FUNCTION_BLOCK FB_ModuleBase EXTENDS FB_PackMLModeSet
VAR_INPUT
	ModuleCtrl : REFERENCE TO ST_ModuleCtrl;
	SystemContext : REFERENCE TO ST_SystemContext;
	HeartbeatIndex : UDINT;
	RuntimeConfig : REFERENCE TO ST_ModuleRuntimeConfig;
	VariableNodeReader : I_VariableNodeReader;
END_VAR

VAR_OUTPUT
	ModuleStatus : ST_ModuleStatus;
	ModuleVariableList : ARRAY[1..Param_Config.MaxModuleVariable] OF ST_ExtDescriptor;
	ModuleAlarmList : ARRAY[1..Param_Config.MaxPublishedModuleAlarms] OF ST_ExtAlarm;
	ModuleDataList : ARRAY[1..Param_Config.MaxModuleData] OF ST_ExtDescriptor;
END_VAR

VAR
	_CmdRequestOneShot : R_TRIG;
	_ModeRequestOneShot : R_TRIG;
	
	_ModuleId : UDINT;
	_ServiceContext : ST_ServiceContext;
	
	_HeartbeatTimer : TON;
	_LastHeartbeatIndex : UDINT;
	_IsControlSourceAlive : BOOL;
	_ConfiguredSnapshot : FB_ConfigValueSnapshotReader;
	_AlarmManager : FB_ModuleAlarmManager;
	_InAlarmHook : BOOL;
	_InVariableHook : BOOL;
	_ConfiguredVariableCount : UINT;
	_ServiceCoordinator : FB_ServiceCoordinator;
	_ServiceRegistrationAttempted : BOOL;
END_VAR

METHOD PROTECTED FINAL H_OnAborting : E_PackMLHookResult
VAR_INPUT
	bFirstScan : BOOL;
END_VAR
H_OnAborting := E_PackMLHookResult.Busy;
IF _ServiceCoordinator.AllAborted THEN
	H_OnAborting := E_PackMLHookResult.Done;
END_IF
END_METHOD

METHOD PROTECTED FINAL H_OnClearing : E_PackMLHookResult
VAR_INPUT
	bFirstScan : BOOL;
END_VAR
H_OnClearing := E_PackMLHookResult.Busy;
IF _ServiceCoordinator.AllStopped THEN
	H_OnClearing := E_PackMLHookResult.Done;
END_IF
END_METHOD

METHOD PROTECTED FINAL H_OnIdle
VAR_INPUT
	bFirstScan	: BOOL;
END_VAR
// Transfer to execute automatically
RequestCommand(E_PackMLCommand.Start);
END_METHOD

METHOD PROTECTED FINAL H_OnResetting : E_PackMLHookResult
VAR_INPUT
	bFirstScan : BOOL;
END_VAR
H_OnResetting := E_PackMLHookResult.Busy;
IF _ServiceCoordinator.AllIdle THEN
	H_OnResetting := E_PackMLHookResult.Done;
END_IF
END_METHOD

METHOD PROTECTED FINAL H_OnStopping : E_PackMLHookResult
VAR_INPUT
	bFirstScan : BOOL;
END_VAR
H_OnStopping := E_PackMLHookResult.Busy;
IF _ServiceCoordinator.AllStopped THEN
	H_OnStopping := E_PackMLHookResult.Done;
END_IF
END_METHOD

METHOD PROTECTED H_RegisterServices
// Derived Modules register persistent Service storage once.
END_METHOD

METHOD PROTECTED H_UpdateAlarm
// Optional Module extension; submitted values belong to this scan.
END_METHOD

METHOD PROTECTED H_UpdateBaseUnit
VAR_INPUT
END_VAR
END_METHOD

METHOD PROTECTED H_UpdateService
VAR_INPUT
END_VAR
END_METHOD

METHOD PROTECTED H_UpdateVariable
// Optional Module extension; submitted values belong to this scan.
END_METHOD

METHOD PROTECTED FINAL M_AddAlarm : BOOL
VAR_INPUT
	MainErrorId : UDINT;
	SourceErrorId : UDINT;
	Message : STRING;
	Path : STRING(255);
	Severity : E_Severity;
END_VAR
VAR
	nIndex : UINT;
	Alarm : ST_ExtAlarm;
END_VAR
M_AddAlarm := FALSE;
IF NOT _InAlarmHook OR (MainErrorId = 0) THEN
	RETURN;
END_IF
IF __ISVALIDREF(RuntimeConfig) THEN
	IF RuntimeConfig.Valid THEN
		FOR nIndex := 1 TO RuntimeConfig.AlarmCount DO
			IF RuntimeConfig.AlarmBindings[nIndex].Definition.MainErrorId = MainErrorId THEN
				M_AddAlarm := TRUE; // JSON owns the complete definition, even without a valid sample.
				RETURN;
			END_IF
		END_FOR
	END_IF
END_IF
MEMSET(ADR(Alarm), 0, SIZEOF(Alarm));
Alarm.MainErrorId := MainErrorId;
Alarm.SourceErrorId := SourceErrorId;
Alarm.Message := Message;
Alarm.Path := Path;
Alarm.Severity := Severity;
Alarm.DateTime := _ServiceContext.UtcDateTime;
M_AddAlarm := _AlarmManager.M_ObserveHookAlarm(Alarm := Alarm);
END_METHOD

METHOD PROTECTED FINAL M_AddVariable : BOOL
VAR_INPUT
	Id : UDINT;
	Name : STRING(30);
	DataType : E_DescriptorType;
	Unit : STRING(10);
	Value : STRING(80);
END_VAR
VAR
	nIndex : UINT;
END_VAR
M_AddVariable := FALSE;
IF NOT _InVariableHook OR (Id = 0) THEN
	RETURN;
END_IF
FOR nIndex := 1 TO ModuleStatus.Variable.PublishedCount DO
	IF ModuleVariableList[nIndex].Id = Id THEN
		IF nIndex <= _ConfiguredVariableCount THEN
			M_AddVariable := TRUE; // JSON ownership is not a duplicate submission.
		ELSIF ModuleStatus.Variable.DuplicateId = 0 THEN
			ModuleStatus.Variable.DuplicateId := Id;
		END_IF
		RETURN;
	END_IF
END_FOR
IF ModuleStatus.Variable.PublishedCount >= Param_Config.MaxModuleVariable THEN
	ModuleStatus.Variable.Overflow := TRUE;
	RETURN;
END_IF
ModuleStatus.Variable.PublishedCount := ModuleStatus.Variable.PublishedCount + 1;
nIndex := ModuleStatus.Variable.PublishedCount;
ModuleVariableList[nIndex].Id := Id;
ModuleVariableList[nIndex].Name := Name;
ModuleVariableList[nIndex].DataType := DataType;
ModuleVariableList[nIndex].Unit := Unit;
ModuleVariableList[nIndex].Value := Value;
M_AddVariable := TRUE;
END_METHOD

METHOD PRIVATE M_CheckHeartbeat
VAR_INPUT
END_VAR

VAR
	bLooseHeartbeat : BOOL;
	HeartbeatTimeout : TIME;
END_VAR
HeartbeatTimeout := SystemContext.ModuleHeartbeatTimeout;
IF HeartbeatTimeout <= T#0S THEN
	HeartbeatTimeout := Param_Config.ModuleHeartbeat_Timeout;
END_IF

// Heartbeats check
bLooseHeartbeat := _LastHeartbeatIndex = HeartbeatIndex;
IF bLooseHeartbeat THEN
	_HeartbeatTimer(IN := TRUE, PT := HeartbeatTimeout);
ELSE
	_HeartbeatTimer(IN := FALSE, PT := HeartbeatTimeout);
END_IF

// Update Last Heartbeat Index
_LastHeartbeatIndex := HeartbeatIndex;

// Update Is ControlSource Alive status
_IsControlSourceAlive := NOT _HeartbeatTimer.Q;
END_METHOD

METHOD PRIVATE M_PublishAlarmState
_AlarmManager.M_Publish(AlarmList := ModuleAlarmList);
ModuleStatus.Alarm.AckResponseId := _AlarmManager.AckResponseId;
ModuleStatus.Alarm.AckAccepted := _AlarmManager.AckAccepted;
ModuleStatus.Alarm.AckError := _AlarmManager.AckError;
ModuleStatus.Alarm.ConfiguredLatchedCount := _AlarmManager.ConfiguredLatchedCount;
ModuleStatus.Alarm.Overflow := _AlarmManager.Overflow;
ModuleStatus.Alarm.ServiceLatchedCount := _AlarmManager.ServiceLatchedCount;
ModuleStatus.Alarm.HookLatchedCount := _AlarmManager.HookLatchedCount;
ModuleStatus.Alarm.DuplicateId := _AlarmManager.DuplicateId;
END_METHOD

METHOD PROTECTED FINAL M_RegisterService : BOOL
VAR_INPUT
	ServiceId : UDINT;
	AllowCompositeCall : BOOL;
	UpperParam : ANY;
	EffectiveParam : ANY;
END_VAR
VAR_IN_OUT
	UpperCtrl : ST_ServiceCtrl;
	EffectiveCtrl : ST_ServiceCtrl;
	Status : ST_ServiceStatus;
END_VAR
M_RegisterService := _ServiceCoordinator.M_Register(
	ServiceId := ServiceId,
	AllowCompositeCall := AllowCompositeCall,
	UpperCtrl := UpperCtrl,
	EffectiveCtrl := EffectiveCtrl,
	UpperParam := UpperParam,
	EffectiveParam := EffectiveParam,
	Status := Status);
END_METHOD

METHOD PRIVATE M_UpdateAlarmState
VAR
	nAlarm : UINT;
	nSource : UINT;
	nRevision : UDINT;
	fValue : LREAL;
	bValid : BOOL;
	bConditionMet : BOOL;
	Alarm : ST_ExtAlarm;
END_VAR
nRevision := 0;
IF __ISVALIDREF(RuntimeConfig) THEN
	IF RuntimeConfig.Valid THEN
		nRevision := RuntimeConfig.Revision;
	END_IF
END_IF
_AlarmManager.M_BeginCycle(
	ModuleId := _ModuleId,
	ConfigurationRevision := nRevision);

// Remove identities now owned by JSON before an acknowledgement can find a stale Hook event.
IF __ISVALIDREF(RuntimeConfig) THEN
	IF RuntimeConfig.Valid THEN
		FOR nAlarm := 1 TO RuntimeConfig.AlarmCount DO
			_AlarmManager.M_SuppressHookAlarm(
				MainErrorId := RuntimeConfig.AlarmBindings[nAlarm].Definition.MainErrorId);
		END_FOR
	END_IF
END_IF

// Process acknowledgements before evaluating this cycle so AckAll cannot consume
// a new event that the upper controller has not observed yet.
_AlarmManager.M_ProcessAcknowledgement(Request := ModuleCtrl.AlarmAckRequest);

IF __ISVALIDREF(RuntimeConfig) THEN
	IF RuntimeConfig.Valid AND _ConfiguredSnapshot.Ready THEN
		FOR nAlarm := 1 TO RuntimeConfig.AlarmCount DO
			nSource := RuntimeConfig.VariableCount + nAlarm;
			fValue := _ConfiguredSnapshot.M_GetLReal(SourceIndex := nSource, Valid => bValid);
			bConditionMet := FALSE;
			IF bValid THEN
				bConditionMet := F_AlarmConditionMet(
					Value := fValue,
					Operator := RuntimeConfig.AlarmBindings[nAlarm].Definition.Operator,
					Threshold := RuntimeConfig.AlarmBindings[nAlarm].Definition.Threshold,
					Tolerance := RuntimeConfig.AlarmBindings[nAlarm].Definition.Tolerance);
			END_IF

			MEMSET(ADR(Alarm), 0, SIZEOF(Alarm));
			Alarm.ModuleId := _ModuleId;
			Alarm.ServiceId := 0;
			Alarm.MainErrorId := RuntimeConfig.AlarmBindings[nAlarm].Definition.MainErrorId;
			Alarm.SourceErrorId := RuntimeConfig.AlarmBindings[nAlarm].Definition.SourceErrorId;
			Alarm.Message := RuntimeConfig.AlarmBindings[nAlarm].Definition.Message;
			Alarm.Path := RuntimeConfig.AlarmBindings[nAlarm].Definition.Source;
			Alarm.Severity := RuntimeConfig.AlarmBindings[nAlarm].Definition.Severity;
			_AlarmManager.M_UpdateConfiguredAlarm(
				AlarmIndex := nAlarm,
				SampleValid := bValid,
				ConditionMet := bConditionMet,
				Alarm := Alarm,
				UtcDateTime := _ServiceContext.UtcDateTime);
		END_FOR
	END_IF
END_IF

_InAlarmHook := TRUE;
H_UpdateAlarm();
_InAlarmHook := FALSE;

M_UpdateServiceAlarms();
_AlarmManager.M_EndCycle();
END_METHOD

METHOD PRIVATE M_UpdateConfiguredVariableList
VAR
	nVariable : UINT;
	bValid : BOOL;
END_VAR
IF NOT __ISVALIDREF(RuntimeConfig) THEN
	RETURN;
END_IF
IF NOT RuntimeConfig.Valid THEN
	RETURN;
END_IF

FOR nVariable := 1 TO RuntimeConfig.VariableCount DO
	ModuleVariableList[nVariable].Id := RuntimeConfig.VariableBindings[nVariable].Definition.Id;
	ModuleVariableList[nVariable].Name := RuntimeConfig.VariableBindings[nVariable].Definition.Name;
	ModuleVariableList[nVariable].DataType := F_ConfigDataTypeToDescriptor(
		DataType := RuntimeConfig.VariableBindings[nVariable].Definition.DataType);
	ModuleVariableList[nVariable].Unit := RuntimeConfig.VariableBindings[nVariable].Definition.Unit;
	ModuleVariableList[nVariable].Value := _ConfiguredSnapshot.M_GetValueString(
		SourceIndex := nVariable,
		Valid => bValid);
END_FOR
_ConfiguredVariableCount := RuntimeConfig.VariableCount;
ModuleStatus.Variable.PublishedCount := _ConfiguredVariableCount;
END_METHOD

METHOD PROTECTED FINAL M_UpdateModule
IF NOT _ServiceRegistrationAttempted THEN
	_ServiceRegistrationAttempted := TRUE;
	_ServiceCoordinator.M_BeginRegistration();
	H_RegisterServices();
	_ServiceCoordinator.M_Seal();
END_IF

M_CheckHeartbeat();
ModuleStatus.IsControlSourceAlive := _IsControlSourceAlive;

// Update module state machine
PackMLIn := ModuleCtrl.PackMLIn;
SUPER^();

IF __ISVALIDREF(RuntimeConfig) THEN
	_ModuleId := RuntimeConfig.ModuleId;
	_ConfiguredSnapshot(
		RuntimeConfig := RuntimeConfig,
		VariableNodeReader := VariableNodeReader);
	ModuleStatus.ModuleId := _ModuleId;
	ModuleStatus.Enabled := RuntimeConfig.Enabled;
	ModuleStatus.ModuleType := RuntimeConfig.ModuleType;
END_IF

_ServiceContext.ModuleId := _ModuleId;
_ServiceContext.UtcDateTime := SystemContext.UtcDateTime;

// Update service state machine
_ServiceCoordinator.M_PrepareCycle(
	ModuleInExecute := PackMLOut.eStateCurrent = E_PackMLState.Execute,
	ModuleCtrl := ModuleCtrl);
H_UpdateService();

// Update base unit state machine
H_UpdateBaseUnit();

// Capture the status set produced by this scan for framework aggregation and
// for the Module PackML transition checks in the next scan.
_ServiceCoordinator.M_ObserveCycle();

_CmdRequestOneShot(CLK:= PackMLIn.bCommandChangeRequest, Q=> );
_ModeRequestOneShot(CLK:= PackMLIn.bModeChangeRequest, Q=> );

// Updata status
IF _CmdRequestOneShot.Q OR _ModeRequestOneShot.Q THEN
	ModuleStatus.ResponseId := ModuleCtrl.RequestId;
END_IF
ModuleStatus.PackMLOut := PackMLOut;

M_UpdateAlarmState();
M_PublishAlarmState();
M_UpdateServiceDataList();
M_UpdateVariableList();
END_METHOD

METHOD PRIVATE M_UpdateServiceAlarms
VAR
	nServiceIndex : UINT;
	nErrorIndex : UINT;
	ServiceStatus : ST_ServiceStatus;
END_VAR
// Submit currently observable Service errors. The manager owns lifecycle state
// and marks identities not observed in this scan inactive during M_EndCycle.
FOR nServiceIndex := 1 TO _ServiceCoordinator.RegisteredCount DO
	IF NOT _ServiceCoordinator.M_GetServiceStatusByIndex(
		Index := nServiceIndex,
		Status => ServiceStatus) THEN
		CONTINUE;
	END_IF
	FOR nErrorIndex := 1 TO Param_Config.MaxServiceError DO
		IF ServiceStatus.ErrorList[nErrorIndex].MainErrorId <> 0 THEN
			_AlarmManager.M_ObserveServiceAlarm(
				Alarm := ServiceStatus.ErrorList[nErrorIndex]);
		END_IF
	END_FOR
END_FOR
END_METHOD

METHOD PRIVATE M_UpdateServiceDataList
VAR
	nServiceIndex : UINT;
	nDataIndex : UINT;
	nPublishedIndex : UINT;
	bDuplicate : BOOL;
	DataId : UDINT;
	ServiceStatus : ST_ServiceStatus;
END_VAR
MEMSET(ADR(ModuleDataList), 0, SIZEOF(ModuleDataList));
MEMSET(ADR(ModuleStatus.Data), 0, SIZEOF(ModuleStatus.Data));

FOR nServiceIndex := 1 TO _ServiceCoordinator.RegisteredCount DO
	IF NOT _ServiceCoordinator.M_GetServiceStatusByIndex(
		Index := nServiceIndex,
		Status => ServiceStatus) THEN
		CONTINUE;
	END_IF
	IF ServiceStatus.Data.Overflow THEN
		ModuleStatus.Data.Overflow := TRUE;
	END_IF

	FOR nDataIndex := 1 TO Param_Config.MaxServiceData DO
		DataId := ServiceStatus.Data.DataList[nDataIndex].Id;
		IF DataId = 0 THEN
			CONTINUE;
		END_IF

		bDuplicate := FALSE;
		FOR nPublishedIndex := 1 TO ModuleStatus.Data.PublishedCount DO
			IF ModuleDataList[nPublishedIndex].Id = DataId THEN
				bDuplicate := TRUE;
				EXIT;
			END_IF
		END_FOR

		IF bDuplicate THEN
			IF ModuleStatus.Data.DuplicateId = 0 THEN
				ModuleStatus.Data.DuplicateId := DataId;
			END_IF
			CONTINUE;
		END_IF

		IF ModuleStatus.Data.PublishedCount >= Param_Config.MaxModuleData THEN
			ModuleStatus.Data.Overflow := TRUE;
			CONTINUE;
		END_IF

		ModuleStatus.Data.PublishedCount := ModuleStatus.Data.PublishedCount + 1;
		ModuleDataList[ModuleStatus.Data.PublishedCount] :=
			ServiceStatus.Data.DataList[nDataIndex];
	END_FOR
END_FOR
END_METHOD

METHOD PRIVATE M_UpdateVariableList
MEMSET(ADR(ModuleVariableList), 0, SIZEOF(ModuleVariableList));
MEMSET(ADR(ModuleStatus.Variable), 0, SIZEOF(ModuleStatus.Variable));
_ConfiguredVariableCount := 0;
M_UpdateConfiguredVariableList();
_InVariableHook := TRUE;
H_UpdateVariable();
_InVariableHook := FALSE;
END_METHOD

END_FUNCTION_BLOCK

(* stored: Version 1.1.0.1, ProductVersion 3.1.4026.18
   POU FB_ModuleBase: Id {6193009a-0dba-45cf-9862-8c04373cb73b}, SpecialFunc None
   Folder HookMethod: Id {0b542957-3892-4df2-b0e7-9c93700d86b5}
   Folder Private: Id {9fe464c1-8082-49c4-bb39-67807fabb98d}
   Folder StateAction: Id {11d8fc2a-f5c5-4f28-ab4c-743399b9bdc9}
   Method H_OnAborting: Id {8915d7ec-4b86-49c6-9413-c27372315251}
   Method H_OnClearing: Id {f0397c47-1f8c-451b-93d5-b31f3f0b03fb}
   Method H_OnIdle: Id {1f951a38-751e-4488-9f76-b0388bffa732}
   Method H_OnResetting: Id {9a955b11-d840-4734-887a-1f112a090756}
   Method H_OnStopping: Id {59c31d14-1773-47ac-a868-c25bd37caf0c}
   Method H_RegisterServices: Id {cfb22052-7349-4b72-a01d-2a1212d3d28d}
   Method H_UpdateAlarm: Id {cb61c708-0f3f-469b-a964-b4b351dc9538}
   Method H_UpdateBaseUnit: Id {cce9c8f5-b668-43c6-ab47-4d2999638c8f}
   Method H_UpdateService: Id {d906a778-6b57-49b8-9e25-ec7461c4759a}
   Method H_UpdateVariable: Id {9d15debf-7709-4c12-8971-2dc378590faa}
   Method M_AddAlarm: Id {7c4e4f34-fc5f-482d-9a72-920e07d0a35d}
   Method M_AddVariable: Id {669b3f9b-b87a-4c72-b049-e0b92818a4d4}
   Method M_CheckHeartbeat: Id {95356be4-c779-4a0a-84d9-ca5fd7d93bc1}
   Method M_PublishAlarmState: Id {055c5419-f6a5-46d2-bb31-19f68a24d121}
   Method M_RegisterService: Id {f7cafede-9912-44aa-8775-3dd24b828568}
   Method M_UpdateAlarmState: Id {6b9b6538-c160-4a7b-93a1-a430b340815a}
   Method M_UpdateConfiguredVariableList: Id {6e5b225f-a33a-409e-827d-1330e9e22088}
   Method M_UpdateModule: Id {a3ee927e-c27b-49bf-8f5e-1ddb1a222fc5}
   Method M_UpdateServiceAlarms: Id {aac9cb3d-dfbb-4fd3-8423-c48f0de4cb6b}
   Method M_UpdateServiceDataList: Id {09acfa8b-205a-4e4b-9f04-1c13883b2574}
   Method M_UpdateVariableList: Id {ae656439-fc0d-4872-8331-77be22b77a2c} *)
